// TIA Portal V16 export
// export: Created 2022-02-04T14:40:20.6022335Z, ExportSetting WithDefaults, DisplayName Totally Integrated Automation Portal, DisplayVersion V16 Update 1, DisplayName TIA Portal Version Control Interface, DisplayVersion V16, DisplayName TIA Portal Openness, DisplayVersion V16, DisplayName SINAMICS Startdrive Advanced, DisplayVersion V16 Update 5, DisplayName SINAMICS Startdrive G130, G150, S120, S150, SINAMICS MV, S210, DisplayVersion V16 Update 5, DisplayName SINAMICS Startdrive G110M, G120, G120C, G120D, G120P, G115D, DisplayVersion V16 Update 5, DisplayName STEP 7 Professional, DisplayVersion V16, DisplayName STEP 7 Safety, DisplayVersion V16, DisplayName WinCC Advanced, DisplayVersion V16, DisplayName SIMATIC Visualization Architect, DisplayVersion V16
DATA_BLOCK "FB_SensLine_DB"   // DB17
AUTHOR : Aspir
VERSION : 0.1
// stored: AutoNumber true, InstanceOfName FB_SensLine, InstanceOfType FB
"FB_SensLine"
   // VAR_INPUT
   //    CutPlankData : Bool;
   //    CollectData : Bool;
   //    ActualChain : Bool;
   //    EnableSensors : Bool;
   //    SensData : Word;
   //    SensQuantity : Int;
   //    MinLength : Int;
   //    SensOffset : Int;
   // END_VAR
   // VAR_OUTPUT
   //    Done : Bool;
   //    Hole : Bool;
   //    Chain : Bool;
   //    Length : Int;
   // END_VAR
   // VAR RETAIN
   //    memento_chain : Bool;
   //    sensor_triggers : Array[0..15] of Bool;
   // END_VAR
BEGIN
END_DATA_BLOCK
